{attribute 'GeneratedUsingTerminal: KL2701'}
{attribute addProperty BoxType "KL2701"}
{attribute addProperty Id "Channel_1AT %Q*Channel_460B8C400"}
{attribute addProperty CRC "3732460390"}
{attribute addProperty Size "0"}
TYPE KL2701_DE78D366 :
STRUCT
	{attribute addProperty Name "Channel_1"}
	Channel_1 : Channel_460B8C40;
END_STRUCT
END_TYPE

(* stored: Version 1.2.0.0, ProductVersion 3.1.4024.9
   DUT KL2701_DE78D366: Id {8a066eb2-6d58-4d65-9399-ba71cd4a6ffe} *)
